# EPICS StreamDevice protocol: iocs/epthallprobe/epthallprobe_serial.proto
#
#  @brief EPICS Stream device protocol file.
#
#  @author Martin Wolfes
#  @date   23.09.2014
#

terminator = LF;

#ExtraInput = Ignore;

read_field {
	out "read";
	in "read %f %*f %*f";
}

read_temp{
	out "temp";
	in "temp %f";
}
